# EPICS autosave request: ADApp/Db/NDAttribute_settings.req
$(P)$(R)AttrName
$(P)$(R)TSNumPoints
$(P)$(R)TSRead.SCAN
